(* IEC 61131-3 sources: CodesysTest/export/SX.dev/Plc Logic/Application/HMIData/Proface/FB_ProfaceInterface.pou, 1 file *)

(* ---- Reset.m.st ---- *)
(*#-#-#-#-#-#-#-#-#-#---Declaration---#-#-#-#-#-#-#-#-#-#-#-#-#*)

METHOD Reset : BOOL
VAR_INPUT
END_VAR
(*#-#-#-#-#-#-#-#-#-#---Implementation---#-#-#-#-#-#-#-#-#-#-#-#-#*)

control.backlightOff := FALSE;
control.buzzerEn := TRUE;
control.buzzerOn := FALSE;
changeScreenNumber := 0;
setDisplay := SCREEN_ON;
